FUNCTION_BLOCK POSTGRE_DB_QUERY
  {SET_ATTRIBUTE(OpcUa, POINT.ENDPOINT)}
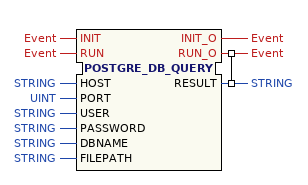
  EVENT_INPUT
    INIT;
    RUN;
  END_EVENT
  EVENT_OUTPUT
    INIT_O;
    RUN_O WITH RESULT;
  END_EVENT
  VAR_INPUT
    HOST : STRING;
    PORT : UINT;
    USER : STRING;
    PASSWORD : STRING;
    DBNAME : STRING;
    FILEPATH : STRING;
  END_VAR
  VAR_OUTPUT
    RESULT : STRING;
  END_VAR
END_FUNCTION_BLOCK
(* other elements stored in the file *)
(* <VarDeclaration Name="RESULT_VALUES" Type="STRING"/> *)
